FUNCTION_BLOCK StackControl
  (* Standard: 61499-2 *)
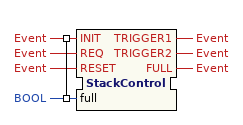
  EVENT_INPUT
    INIT WITH full;
    REQ;
    RESET;
  END_EVENT
  EVENT_OUTPUT
    TRIGGER1;
    TRIGGER2;
    FULL;
  END_EVENT
  VAR_INPUT
    full : BOOL;
  END_VAR
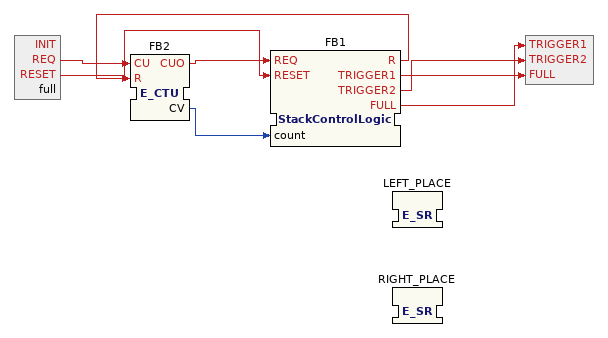
  FBS
    FB1 : StackControlLogic;
    FB2 : E_CTU;
    LEFT_PLACE : E_SR;
    RIGHT_PLACE : E_SR;
  END_FBS
  EVENT_CONNECTIONS
    FB2.CUO TO FB1.REQ;
    REQ TO FB2.CU;
    RESET TO FB1.RESET;
    FB1.R TO FB2.R;
    FB1.TRIGGER1 TO TRIGGER1;
    FB1.TRIGGER2 TO TRIGGER2;
    FB1.FULL TO FULL;
  END_CONNECTIONS
  DATA_CONNECTIONS
    FB2.CV TO FB1.count;
  END_CONNECTIONS
END_FUNCTION_BLOCK
